(* LS Electric XG5000 project: project3 *)
(* PLC LSPLC *)

FUNCTION_BLOCK 위치사용
VAR_INPUT
    s11 : BOOL;
    s12 : BOOL;
    s13 : BOOL;
    s21 : BOOL;
    s22 : BOOL;
    s23 : BOOL;
    s31 : BOOL;
    s32 : BOOL;
    s33 : BOOL;
END_VAR
VAR_OUTPUT
    out11 : WORD;
    out12 : WORD;
    out13 : WORD;
    out21 : WORD;
    out22 : WORD;
    out23 : WORD;
    out31 : WORD;
    out32 : WORD;
    out33 : WORD;
END_VAR
VAR
    mout11 : INT;
    mout12 : INT;
    mout13 : INT;
    mout21 : INT;
    mout22 : INT;
    mout23 : INT;
    mout31 : INT;
    mout32 : INT;
    mout33 : INT;
END_VAR
VAR
    _e1 : R_TRIG;
    _e2 : F_TRIG;
    _e3 : R_TRIG;
    _e4 : F_TRIG;
    _e5 : R_TRIG;
    _e6 : F_TRIG;
    _e7 : R_TRIG;
    _e8 : F_TRIG;
    _e9 : R_TRIG;
    _e10 : F_TRIG;
    _e11 : R_TRIG;
    _e12 : F_TRIG;
    _e13 : R_TRIG;
    _e14 : F_TRIG;
    _e15 : R_TRIG;
    _e16 : F_TRIG;
    _e17 : R_TRIG;
    _e18 : F_TRIG;
END_VAR

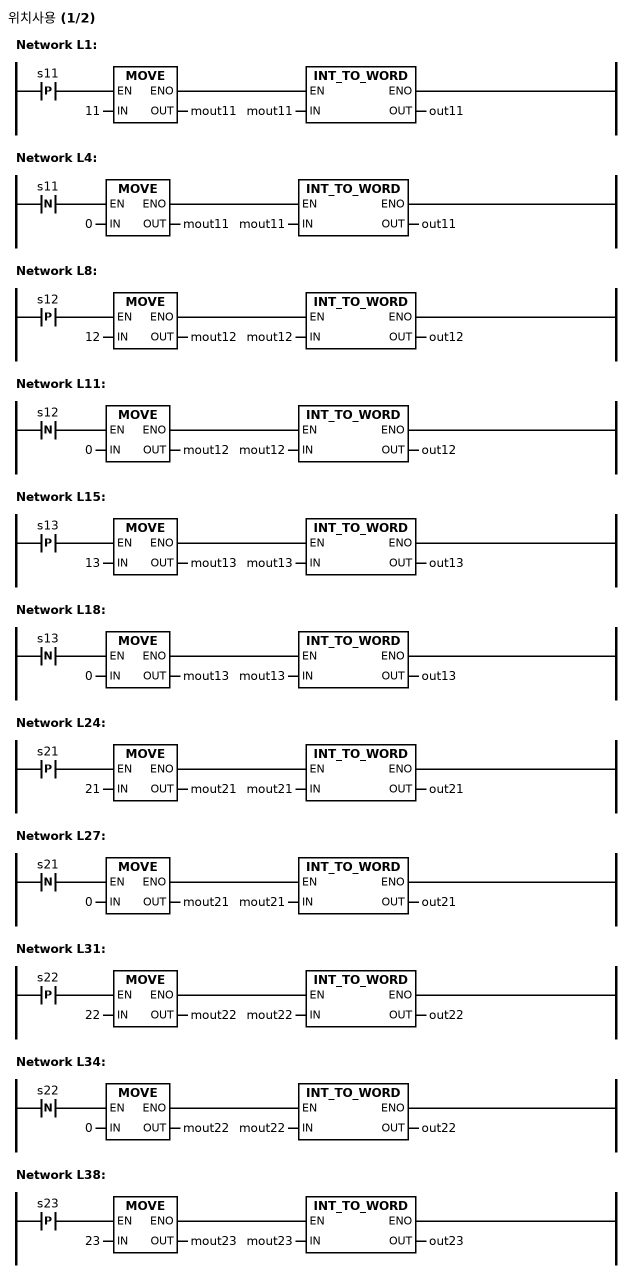
(* Rung L1 *)
_e1(CLK := s11);
IF _e1.Q THEN
    mout11 := 11;
    out11 := INT_TO_WORD(mout11);
END_IF;
(* Rung L4 *)
_e2(CLK := s11);
IF _e2.Q THEN
    mout11 := 0;
    out11 := INT_TO_WORD(mout11);
END_IF;
(* Rung L8 *)
_e3(CLK := s12);
IF _e3.Q THEN
    mout12 := 12;
    out12 := INT_TO_WORD(mout12);
END_IF;
(* Rung L11 *)
_e4(CLK := s12);
IF _e4.Q THEN
    mout12 := 0;
    out12 := INT_TO_WORD(mout12);
END_IF;
(* Rung L15 *)
_e5(CLK := s13);
IF _e5.Q THEN
    mout13 := 13;
    out13 := INT_TO_WORD(mout13);
END_IF;
(* Rung L18 *)
_e6(CLK := s13);
IF _e6.Q THEN
    mout13 := 0;
    out13 := INT_TO_WORD(mout13);
END_IF;
(* Rung L24 *)
_e7(CLK := s21);
IF _e7.Q THEN
    mout21 := 21;
    out21 := INT_TO_WORD(mout21);
END_IF;
(* Rung L27 *)
_e8(CLK := s21);
IF _e8.Q THEN
    mout21 := 0;
    out21 := INT_TO_WORD(mout21);
END_IF;
(* Rung L31 *)
_e9(CLK := s22);
IF _e9.Q THEN
    mout22 := 22;
    out22 := INT_TO_WORD(mout22);
END_IF;
(* Rung L34 *)
_e10(CLK := s22);
IF _e10.Q THEN
    mout22 := 0;
    out22 := INT_TO_WORD(mout22);
END_IF;
(* Rung L38 *)
_e11(CLK := s23);
IF _e11.Q THEN
    mout23 := 23;
    out23 := INT_TO_WORD(mout23);
END_IF;

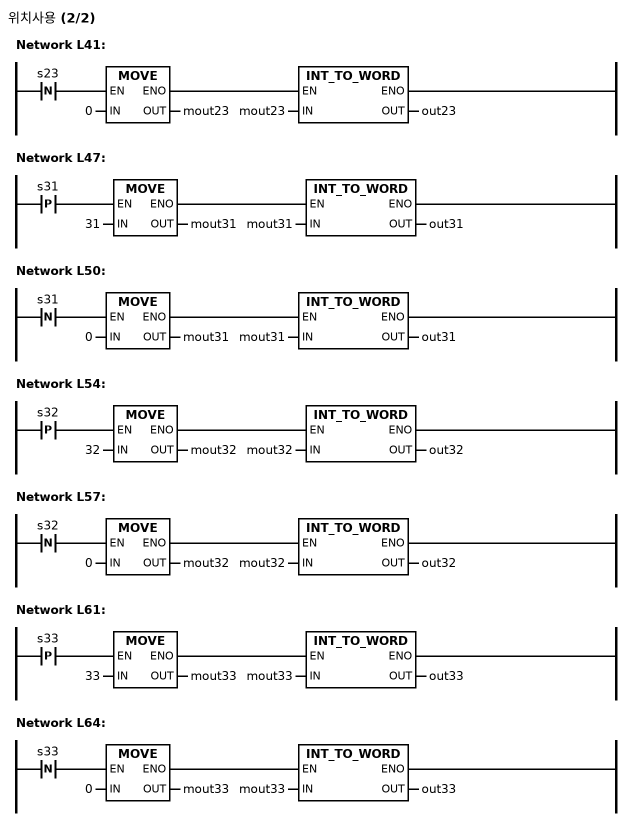
(* Rung L41 *)
_e12(CLK := s23);
IF _e12.Q THEN
    mout23 := 0;
    out23 := INT_TO_WORD(mout23);
END_IF;
(* Rung L47 *)
_e13(CLK := s31);
IF _e13.Q THEN
    mout31 := 31;
    out31 := INT_TO_WORD(mout31);
END_IF;
(* Rung L50 *)
_e14(CLK := s31);
IF _e14.Q THEN
    mout31 := 0;
    out31 := INT_TO_WORD(mout31);
END_IF;
(* Rung L54 *)
_e15(CLK := s32);
IF _e15.Q THEN
    mout32 := 32;
    out32 := INT_TO_WORD(mout32);
END_IF;
(* Rung L57 *)
_e16(CLK := s32);
IF _e16.Q THEN
    mout32 := 0;
    out32 := INT_TO_WORD(mout32);
END_IF;
(* Rung L61 *)
_e17(CLK := s33);
IF _e17.Q THEN
    mout33 := 33;
    out33 := INT_TO_WORD(mout33);
END_IF;
(* Rung L64 *)
_e18(CLK := s33);
IF _e18.Q THEN
    mout33 := 0;
    out33 := INT_TO_WORD(mout33);
END_IF;
END_FUNCTION_BLOCK

FUNCTION_BLOCK 초기화
VAR_INPUT
    초기화 : BOOL;
END_VAR
VAR_OUTPUT
    출력 : BOOL;
END_VAR
VAR
    INST1 : TON;
    INST2 : TP;
END_VAR

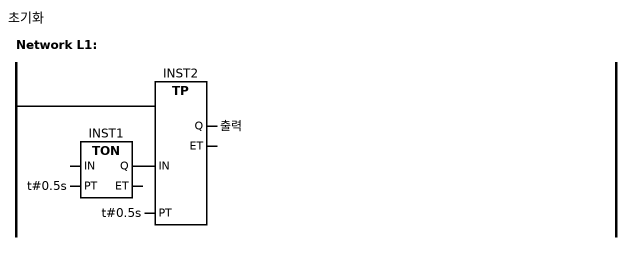
(* Rung L1 *)
INST1(IN := TRUE, PT := t#0.5s);
INST2(IN := INST1.Q, PT := t#0.5s, Q => 출력);
END_FUNCTION_BLOCK

FUNCTION_BLOCK move11
VAR_INPUT
    auto : BOOL;
END_VAR
VAR_OUTPUT
    move11 : BOOL; (* 11 *)
    move21 : BOOL; (* 21 *)
    move31 : BOOL; (* 31 *)
    move32 : BOOL; (* 32 *)
    move33 : BOOL; (* 33 *)
END_VAR
VAR
    X1 : TON;
    X2 : TON;
    X3 : TON;
    Y1 : TON;
    Y2 : TON;
END_VAR

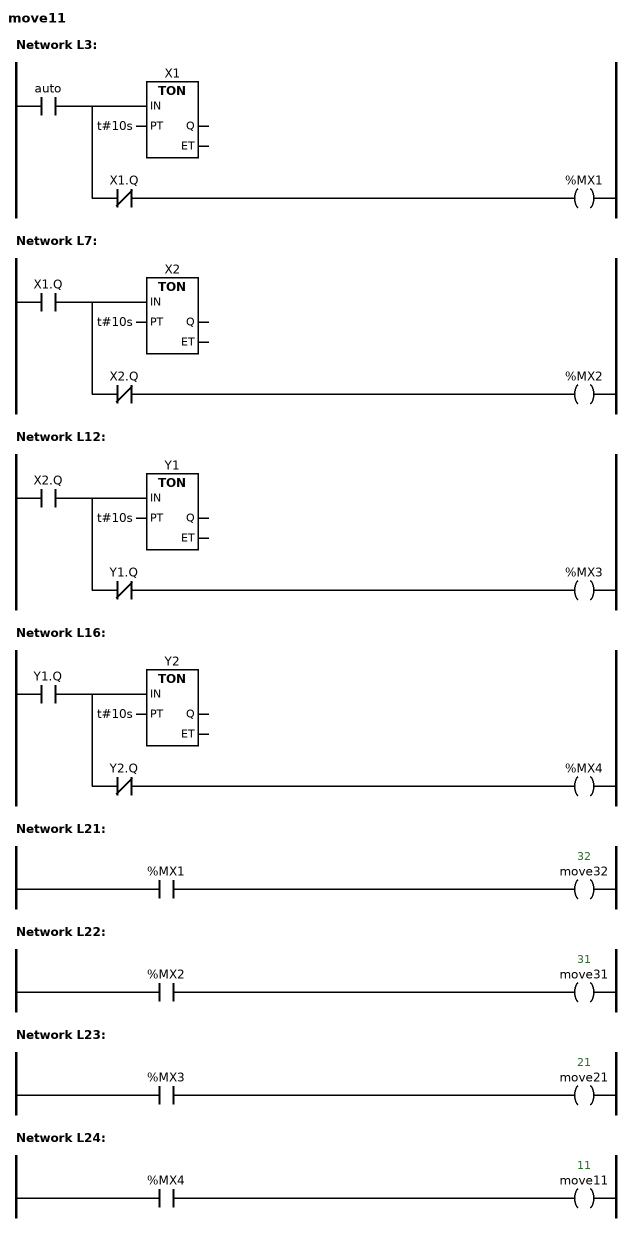
(* Rung L3 *)
X1(IN := auto, PT := t#10s);
%MX1 := auto AND NOT X1.Q;
(* Rung L7 *)
X2(IN := X1.Q, PT := t#10s);
%MX2 := X1.Q AND NOT X2.Q;
(* Rung L12 *)
Y1(IN := X2.Q, PT := t#10s);
%MX3 := X2.Q AND NOT Y1.Q;
(* Rung L16 *)
Y2(IN := Y1.Q, PT := t#10s);
%MX4 := Y1.Q AND NOT Y2.Q;
(* Rung L21 *)
move32 := %MX1;
(* Rung L22 *)
move31 := %MX2;
(* Rung L23 *)
move21 := %MX3;
(* Rung L24 *)
move11 := %MX4;
END_FUNCTION_BLOCK

FUNCTION_BLOCK move12
VAR_INPUT
    auto : BOOL;
END_VAR
VAR
    move12 : BOOL; (* 12 *)
    move22 : BOOL; (* 22 *)
    move32 : BOOL; (* 32 *)
    X1 : TON;
    X2 : TON;
    Y1 : TON;
    Y2 : TON;
END_VAR

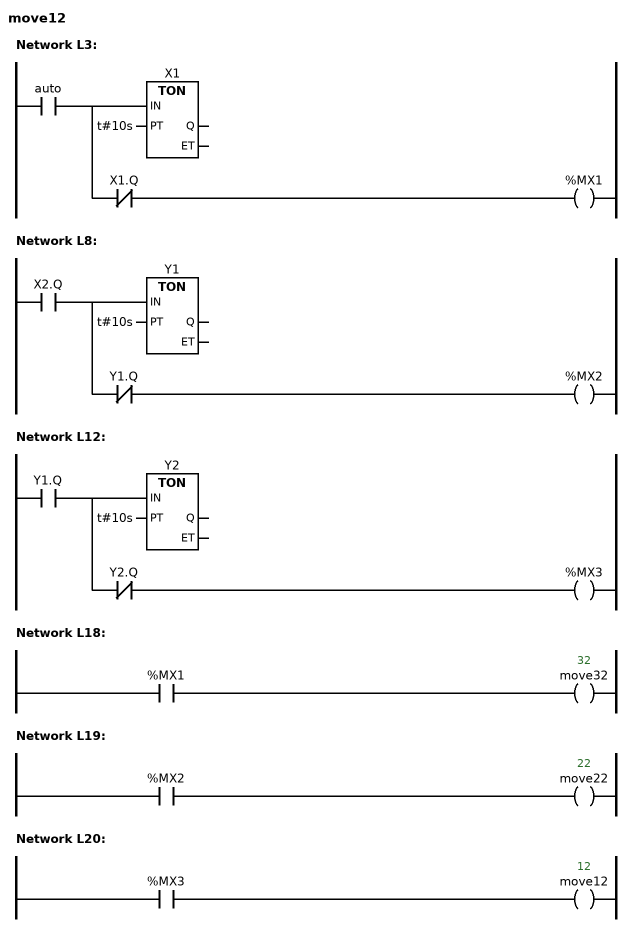
(* Rung L3 *)
X1(IN := auto, PT := t#10s);
%MX1 := auto AND NOT X1.Q;
(* Rung L8 *)
Y1(IN := X2.Q, PT := t#10s);
%MX2 := X2.Q AND NOT Y1.Q;
(* Rung L12 *)
Y2(IN := Y1.Q, PT := t#10s);
%MX3 := Y1.Q AND NOT Y2.Q;
(* Rung L18 *)
move32 := %MX1;
(* Rung L19 *)
move22 := %MX2;
(* Rung L20 *)
move12 := %MX3;
END_FUNCTION_BLOCK

FUNCTION_BLOCK move13
VAR_INPUT
    auto : BOOL;
END_VAR
VAR_OUTPUT
    move33 : BOOL; (* 33 *)
    move32 : BOOL; (* 32 *)
    move22 : BOOL;
    move12 : BOOL;
END_VAR
VAR
    move13 : BOOL; (* 13 *)
    move23 : BOOL; (* 23 *)
    X1 : TON;
    X2 : TON;
    Y1 : TON;
    Y2 : TON;
END_VAR

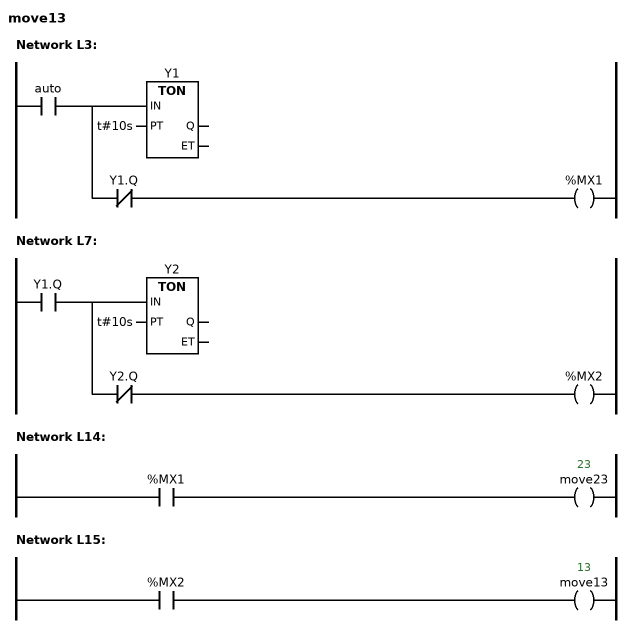
(* Rung L3 *)
Y1(IN := auto, PT := t#10s);
%MX1 := auto AND NOT Y1.Q;
(* Rung L7 *)
Y2(IN := Y1.Q, PT := t#10s);
%MX2 := Y1.Q AND NOT Y2.Q;
(* Rung L14 *)
move23 := %MX1;
(* Rung L15 *)
move13 := %MX2;
END_FUNCTION_BLOCK

PROGRAM NewProgram (* task: 스캔 프로그램 *)
VAR
    A AT %QX0.2.0 : BOOL;
    a1 : ARRAY[0..9] OF INT;
    AD : BOOL := 0;
    A_check AT %QX0.5.0 : BOOL;
    A_delay : TON;
    A_delay_유지 : BOOL;
    A_last : TON;
    A_pull : BOOL;
    A_push : BOOL;
    A_way AT %QX0.6.0 : BOOL;
    A단락 : BOOL;
    A센서 AT %QX0.9.0 : BOOL; (* 센서 *)
    A센서_딜레이 : TON;
    A센서상태변경 : TON;
    A센서지연 : TON;
    A센서지연1 : TON;
    A실린더_OFF AT %IX0.1.1 : BOOL; (* 실린더 *)
    A실린더_ON AT %IX0.1.0 : BOOL; (* 실린더 *)
    A지연 : TON;
    A차단 : TON;
    A카운트 : CTU_INT;
    A타이머 : TON;
    B AT %QX0.2.1 : BOOL;
    BD : BOOL := 0;
    B_check AT %QX0.5.1 : BOOL;
    B_delay : TON;
    B_delay_유지 : BOOL;
    B_last : TON;
    b_pull : BOOL;
    B_push : BOOL;
    B_way AT %QX0.6.1 : BOOL;
    B단락 : BOOL;
    B센서 AT %QX0.9.1 : BOOL; (* 센서 *)
    B센서_딜레이 : TON;
    B센서상태변경 : TON;
    B센서지연 : TON;
    B센서지연1 : TON;
    B실린더_OFF AT %IX0.1.3 : BOOL; (* 실린더 *)
    B실린더_ON AT %IX0.1.2 : BOOL; (* 실린더 *)
    B지연 : TON;
    B차단 : TON;
    B카운트 : CTU_INT;
    B타이머 : TON;
    C AT %QX0.2.2 : BOOL;
    CD : BOOL := 0;
    CU : BOOL;
    C_check AT %QX0.5.2 : BOOL;
    C_delay : TON;
    C_delay_유지 : BOOL;
    C_last : TON;
    c_out : BOOL;
    C_pull : BOOL;
    C_push : BOOL;
    C_way AT %QX0.6.2 : BOOL;
    C단락 : BOOL;
    C센서 AT %QX0.9.2 : BOOL; (* 센서 *)
    C센서_딜레이 : TON;
    C센서상태변경 : TON;
    C센서지연 : TON;
    C센서지연1 : TON;
    C실린더_OFF AT %IX0.1.5 : BOOL; (* 실린더 *)
    C실린더_ON AT %IX0.1.4 : BOOL; (* 실린더 *)
    C지연 : TON;
    C차단 : TON;
    C카운트 : CTUD_INT;
    C카운트1 : CTUD_INT;
    C타이머 : TON;
    C타이머1 : TON;
    C타이머2 : TON;
    D1 : WORD;
    D91 : TIME;
    delay : TP;
    done : BOOL;
    d_a AT %IW0.3.0 : WORD;
    d_a_out : UDINT;
    d_a_time : TIME;
    d_b AT %IW0.3.1 : WORD;
    d_b_out : UDINT;
    d_b_time : TIME;
    d_input : BOOL;
    ET : TIME;
    fifo : FIFO_INT;
    INST : TP;
    INST1 : TP;
    INST10 : TP;
    INST11 : TP;
    INST12 : TP;
    INST13 : TP;
    INST14 : TP;
    INST15 : TP;
    INST16 : TP;
    INST17 : TP;
    INST18 : TP;
    INST19 : TP;
    INST2 : TP;
    INST20 : TP;
    INST21 : TP;
    INST22 : TP;
    INST23 : TP;
    INST24 : TP;
    INST25 : TP;
    INST26 : TP;
    INST27 : TP;
    INST28 : TP;
    INST29 : TP;
    INST3 : TP;
    INST30 : TP;
    INST31 : TP;
    INST32 : TP;
    INST33 : TP;
    INST34 : TP;
    INST35 : TP;
    INST36 : TP;
    INST37 : TP;
    INST38 : CTUD_INT;
    INST4 : TP;
    INST5 : TP;
    INST6 : TP;
    INST7 : TP;
    INST8 : TP;
    INST9 : TP;
    LD : BOOL;
    LOAD : BOOL;
    OUT AT %QW0.8.0 : INT;
    output1 : INT;
    output2 : UDINT;
    output3 : INT;
    output4 : UDINT;
    output5 : INT;
    output6 : UDINT;
    output7 : INT;
    output8 : UDINT;
    prev AT %QW0.8.1 : WORD;
    prev_int : INT;
    PV : INT;
    QD : BOOL;
    QU : BOOL;
    R : BOOL;
    rand : INT;
    reset : BOOL;
    RST : BOOL;
    s11 : BOOL;
    s12 : BOOL;
    s13 : BOOL;
    s21 : BOOL;
    s22 : BOOL;
    s23 : BOOL;
    s31 : BOOL;
    s32 : BOOL;
    s33 : BOOL;
    set : BOOL;
    signal : BOOL;
    stack : CTUD_INT;
    stack_max : INT := 9; (* max *)
    stack_센서 : BOOL;
    stack센서 : BOOL;
    start : BOOL;
    stop AT %IX0.0.1 : BOOL;
    system_on AT %IX0.0.0 : BOOL;
    temp AT %IX0.0.2 : BOOL;
    test1 : BOOL;
    test2 : BOOL;
    three : WORD := 3;
    time1 : TIME;
    time2 : TIME;
    time3 : TIME;
    time4 : TIME;
    UNLD : BOOL;
    X1 : TON;
    X2 : TON;
    X3 : TON;
    Y1 : TON;
    Y2 : TON;
    Y3 : TON;
    _T15S : BOOL;
    긴급제동 : BOOL; (* RED *)
    난수1 : TON;
    난수2 : TON;
    난수회로차단 : TP;
    놓기 AT %QX0.0.49 : BOOL;
    단선 AT %QX0.8.1 : BOOL;
    도착 AT %QX0.5.3 : BOOL;
    딜레이 : TON;
    랜덤수 : INT;
    명령 : BOOL;
    물품없음 : BOOL; (* WHITE *)
    반시계 AT %QX0.0.62 : BOOL;
    백색등 : BOOL;
    상 AT %QX0.0.60 : BOOL;
    선택값 : INT;
    소요시간1 : TIME;
    수동 : BOOL;
    순환값 : WORD;
    숫자 : INT := 1;
    시계 AT %QX0.0.61 : BOOL;
    시퀀스1 AT %MW4 : INT;
    시퀀스2 AT %MW8 : INT;
    신호 AT %QX0.6.3 : BOOL;
    앞 AT %QX0.0.59 : BOOL;
    연기 : BOOL;
    위치사용 : 위치사용;
    임시 : BOOL;
    입고 : CTUD_INT;
    입력 : BOOL;
    입력1 AT %QX0.6.4 : BOOL;
    입력시간1 AT %MW6 : INT;
    입력시간2 AT %MW2 : INT;
    입력시간3 AT %MW10 : INT;
    입력시간4 AT %MW12 : INT;
    입력신호 AT %QW0.6.3 : INT;
    자동 : BOOL;
    잡기 AT %QX0.0.63 : BOOL;
    저장 : FIFO_INT;
    정상가동 : BOOL; (* GREEN *)
    지연 : TON;
    지연1 : TP;
    초기화 : 초기화;
    출력 : BOOL;
    칸1 AT %QX0.0.50 : BOOL;
    칸10 AT %QX0.0.44 : BOOL;
    칸11 AT %QX0.0.47 : BOOL;
    칸12 AT %QX0.0.46 : BOOL;
    칸2 AT %QX0.0.51 : BOOL;
    칸3 AT %QX0.0.52 : BOOL;
    칸4 AT %QX0.0.53 : BOOL;
    칸5 AT %QX0.0.54 : BOOL;
    칸6 AT %QX0.0.55 : BOOL;
    칸7 AT %QX0.0.56 : BOOL;
    칸8 AT %QX0.0.57 : BOOL;
    칸9 AT %QX0.0.58 : BOOL;
    컨베이어벨트 AT %QX0.4.4 : BOOL;
    컨베이어타이머 : TON;
    하 AT %QX0.0.45 : BOOL;
    하나출력 : BOOL;
END_VAR
VAR
    _t1 : BOOL;
    _e2 : R_TRIG;
    _e3 : F_TRIG;
    _e4 : F_TRIG;
    _e5 : F_TRIG;
    _e6 : F_TRIG;
    _e7 : R_TRIG;
    _e8 : R_TRIG;
    _p9 : BOOL;
    _p10 : BOOL;
    _e11 : R_TRIG;
    _p12 : BOOL;
    _p13 : BOOL;
    _e14 : R_TRIG;
    _p15 : BOOL;
    _p16 : BOOL;
    _e17 : R_TRIG;
    _p18 : BOOL;
    _e19 : R_TRIG;
    _e20 : R_TRIG;
    _e21 : R_TRIG;
    _t22 : BOOL;
    _e23 : F_TRIG;
    _e24 : F_TRIG;
    _e25 : F_TRIG;
    _e26 : F_TRIG;
    _e27 : F_TRIG;
    _e28 : F_TRIG;
    _e29 : F_TRIG;
    _e30 : F_TRIG;
    _e31 : F_TRIG;
    _e32 : F_TRIG;
    _e33 : F_TRIG;
    _e34 : F_TRIG;
    _e35 : F_TRIG;
    _e36 : F_TRIG;
    _e37 : F_TRIG;
    _e38 : F_TRIG;
    _e39 : F_TRIG;
    _e40 : F_TRIG;
    _e41 : F_TRIG;
    _e42 : F_TRIG;
    _e43 : F_TRIG;
    _e44 : F_TRIG;
    _e45 : F_TRIG;
    _e46 : F_TRIG;
    _e47 : F_TRIG;
    _e48 : F_TRIG;
    _e49 : F_TRIG;
    _e50 : F_TRIG;
    _e51 : F_TRIG;
    _e52 : F_TRIG;
    _e53 : F_TRIG;
    _e54 : F_TRIG;
    _e55 : F_TRIG;
    _e56 : F_TRIG;
    _e57 : F_TRIG;
    _e58 : F_TRIG;
    _e59 : F_TRIG;
    _e60 : F_TRIG;
    _e61 : F_TRIG;
END_VAR

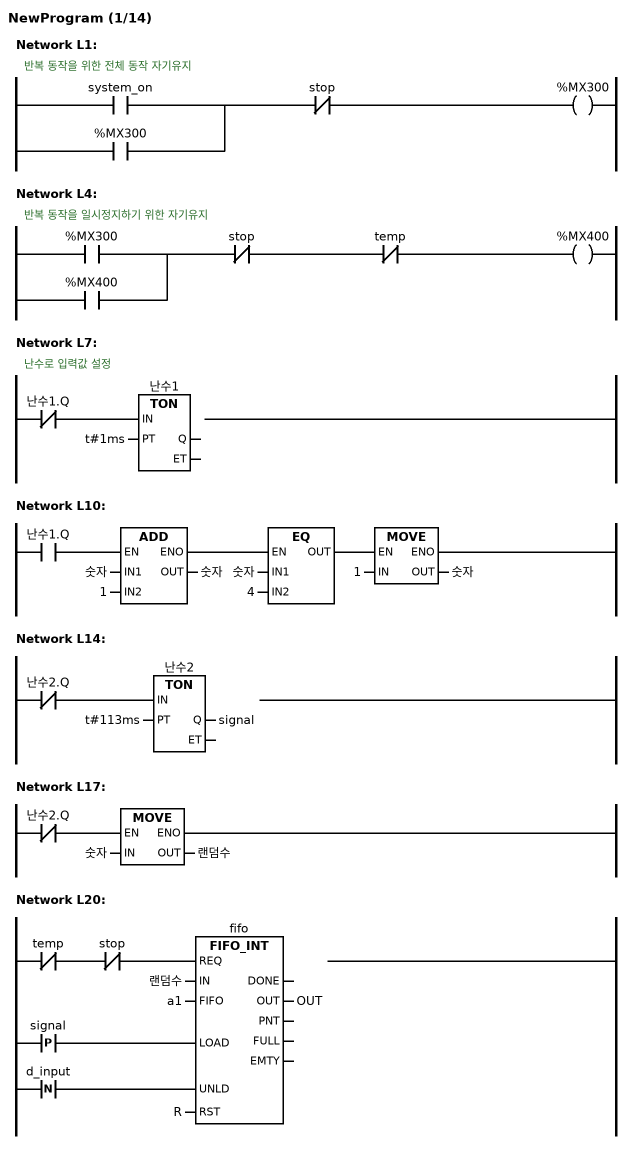
(* 반복 동작을 위한 전체 동작 자기유지 *)
(* Rung L1 *)
%MX300 := (system_on OR %MX300) AND NOT stop;
(* 반복 동작을 일시정지하기 위한 자기유지 *)
(* Rung L4 *)
%MX400 := (%MX300 OR %MX400) AND NOT stop AND NOT temp;
(* 난수로 입력값 설정 *)
(* Rung L7 *)
난수1(IN := NOT 난수1.Q, PT := t#1ms);
(* Rung L10 *)
IF 난수1.Q THEN
    숫자 := 숫자 + 1;
    _t1 := 숫자 = 4;
END_IF;
IF _t1 THEN 숫자 := 1; END_IF;
(* Rung L14 *)
난수2(IN := NOT 난수2.Q, PT := t#113ms, Q => signal);
(* Rung L17 *)
IF NOT 난수2.Q THEN 랜덤수 := 숫자; END_IF;
(* Rung L20 *)
_e2(CLK := signal);
_e3(CLK := d_input);
fifo(REQ := NOT temp AND NOT stop, IN := 랜덤수, FIFO := a1, LOAD := _e2.Q, UNLD := _e3.Q, RST := R, OUT => OUT);

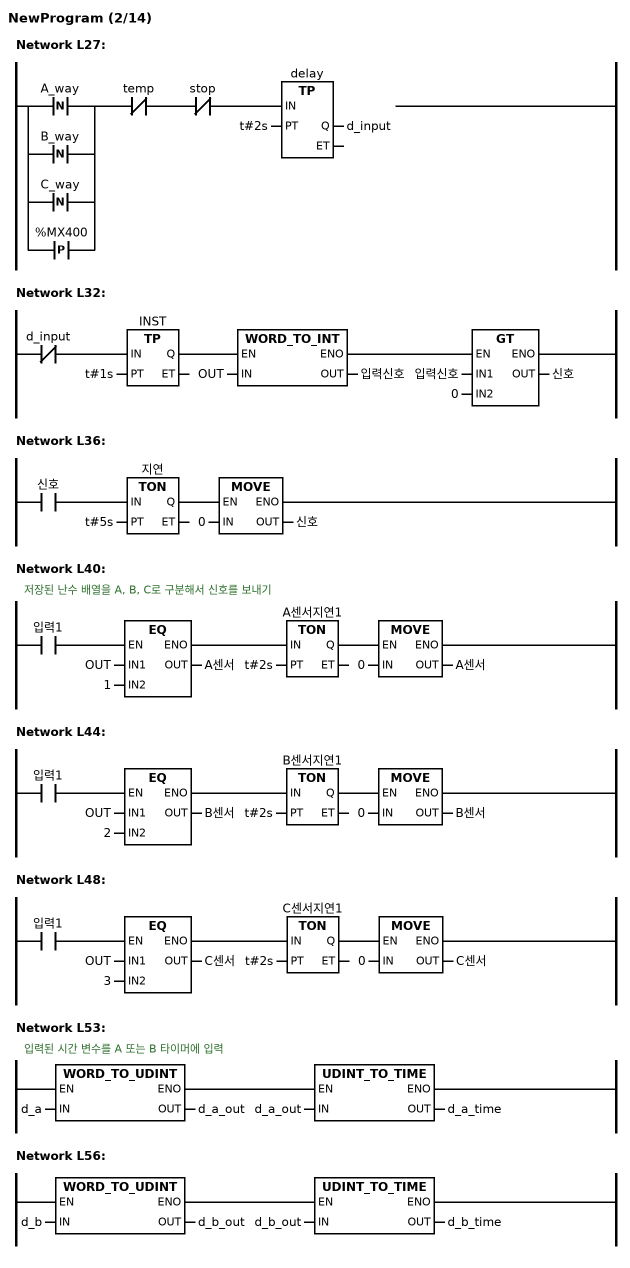
(* Rung L27 *)
_e4(CLK := A_way);
_e5(CLK := B_way);
_e6(CLK := C_way);
_e7(CLK := %MX400);
delay(IN := (_e4.Q OR _e5.Q OR _e6.Q OR _e7.Q) AND NOT temp AND NOT stop, PT := t#2s, Q => d_input);
(* Rung L32 *)
INST(IN := NOT d_input, PT := t#1s);
IF INST.Q THEN
    입력신호 := WORD_TO_INT(OUT);
    신호 := 입력신호 > 0;
END_IF;
(* Rung L36 *)
지연(IN := 신호, PT := t#5s);
IF 지연.Q THEN 신호 := 0; END_IF;
(* 저장된 난수 배열을 A, B, C로 구분해서 신호를 보내기 *)
(* Rung L40 *)
IF 입력1 THEN A센서 := OUT = 1; END_IF;
A센서지연1(IN := 입력1, PT := t#2s);
IF A센서지연1.Q THEN A센서 := 0; END_IF;
(* Rung L44 *)
IF 입력1 THEN B센서 := OUT = 2; END_IF;
B센서지연1(IN := 입력1, PT := t#2s);
IF B센서지연1.Q THEN B센서 := 0; END_IF;
(* Rung L48 *)
IF 입력1 THEN C센서 := OUT = 3; END_IF;
C센서지연1(IN := 입력1, PT := t#2s);
IF C센서지연1.Q THEN C센서 := 0; END_IF;
(* 입력된 시간 변수를 A 또는 B 타이머에 입력 *)
(* Rung L53 *)
d_a_out := WORD_TO_UDINT(d_a);
d_a_time := UDINT_TO_TIME(d_a_out);
(* Rung L56 *)
d_b_out := WORD_TO_UDINT(d_b);
d_b_time := UDINT_TO_TIME(d_b_out);

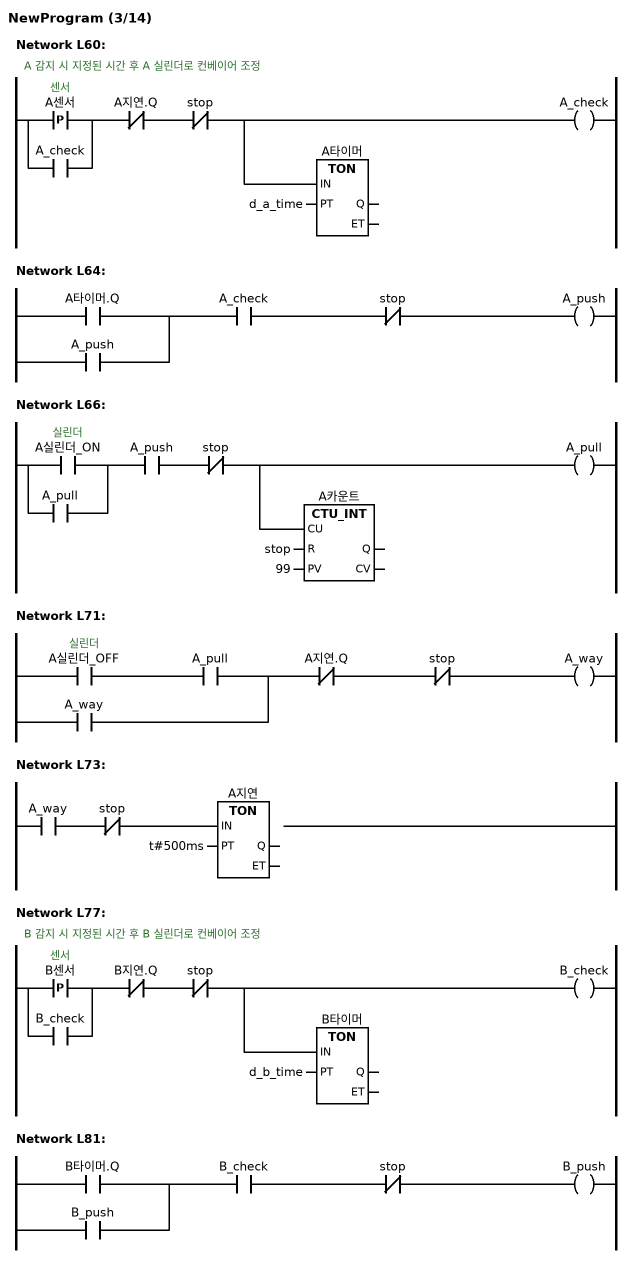
(* A 감지 시 지정된 시간 후 A 실린더로 컨베이어 조정 *)
(* Rung L60 *)
_e8(CLK := A센서);
_p9 := (_e8.Q OR A_check) AND NOT A지연.Q AND NOT stop;
A_check := _p9;
A타이머(IN := _p9, PT := d_a_time);
(* Rung L64 *)
A_push := (A타이머.Q OR A_push) AND A_check AND NOT stop;
(* Rung L66 *)
_p10 := (A실린더_ON OR A_pull) AND A_push AND NOT stop;
A_pull := _p10;
A카운트(CU := _p10, R := stop, PV := 99);
(* Rung L71 *)
A_way := ((A실린더_OFF AND A_pull) OR A_way) AND NOT A지연.Q AND NOT stop;
(* Rung L73 *)
A지연(IN := A_way AND NOT stop, PT := t#500ms);
(* B 감지 시 지정된 시간 후 B 실린더로 컨베이어 조정 *)
(* Rung L77 *)
_e11(CLK := B센서);
_p12 := (_e11.Q OR B_check) AND NOT B지연.Q AND NOT stop;
B_check := _p12;
B타이머(IN := _p12, PT := d_b_time);
(* Rung L81 *)
B_push := (B타이머.Q OR B_push) AND B_check AND NOT stop;

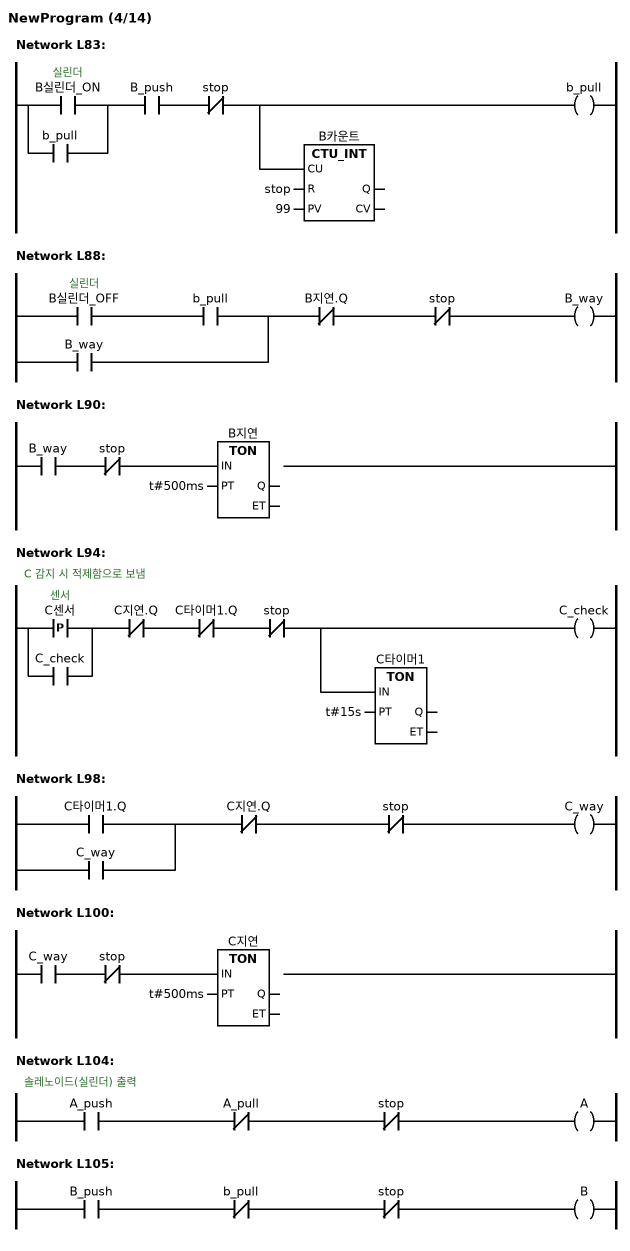
(* Rung L83 *)
_p13 := (B실린더_ON OR b_pull) AND B_push AND NOT stop;
b_pull := _p13;
B카운트(CU := _p13, R := stop, PV := 99);
(* Rung L88 *)
B_way := ((B실린더_OFF AND b_pull) OR B_way) AND NOT B지연.Q AND NOT stop;
(* Rung L90 *)
B지연(IN := B_way AND NOT stop, PT := t#500ms);
(* C 감지 시 적제함으로 보냄 *)
(* Rung L94 *)
_e14(CLK := C센서);
_p15 := (_e14.Q OR C_check) AND NOT C지연.Q AND NOT C타이머1.Q AND NOT stop;
C_check := _p15;
C타이머1(IN := _p15, PT := t#15s);
(* Rung L98 *)
C_way := (C타이머1.Q OR C_way) AND NOT C지연.Q AND NOT stop;
(* Rung L100 *)
C지연(IN := C_way AND NOT stop, PT := t#500ms);
(* 솔레노이드(실린더) 출력 *)
(* Rung L104 *)
A := A_push AND NOT A_pull AND NOT stop;
(* Rung L105 *)
B := B_push AND NOT b_pull AND NOT stop;

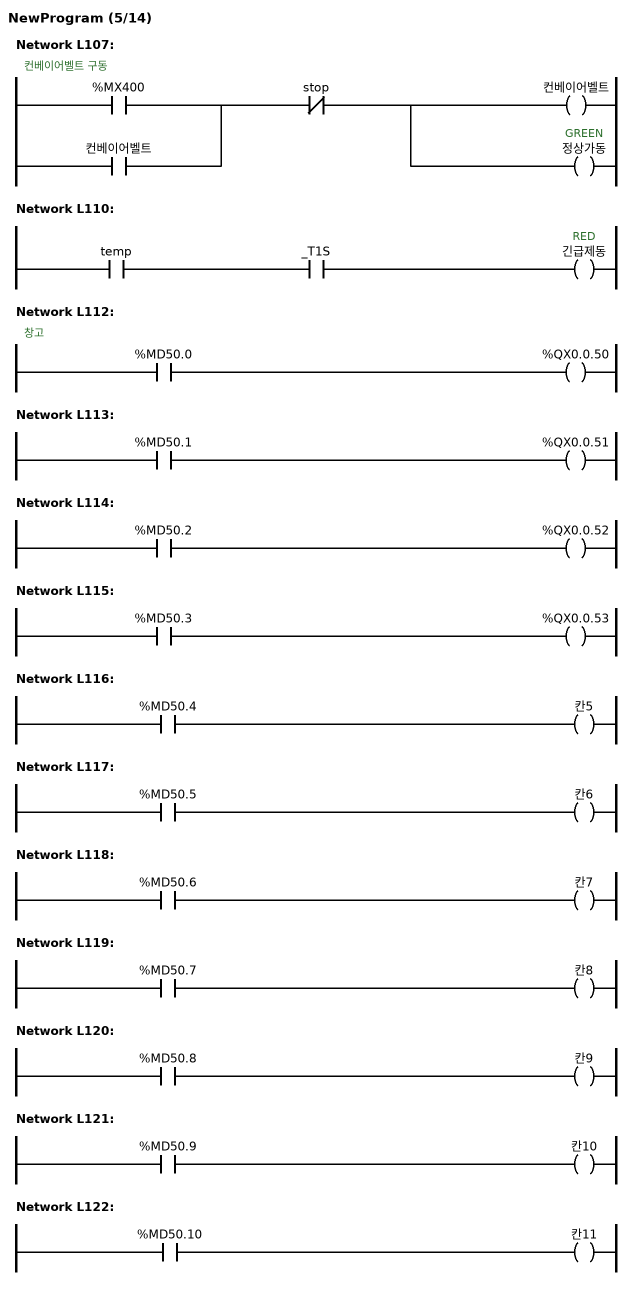
(* 컨베이어벨트 구동 *)
(* Rung L107 *)
_p16 := (%MX400 OR 컨베이어벨트) AND NOT stop;
컨베이어벨트 := _p16;
정상가동 := _p16;
(* Rung L110 *)
긴급제동 := temp AND _T1S;
(* 창고 *)
(* Rung L112 *)
%QX0.0.50 := %MD50.0;
(* Rung L113 *)
%QX0.0.51 := %MD50.1;
(* Rung L114 *)
%QX0.0.52 := %MD50.2;
(* Rung L115 *)
%QX0.0.53 := %MD50.3;
(* Rung L116 *)
칸5 := %MD50.4;
(* Rung L117 *)
칸6 := %MD50.5;
(* Rung L118 *)
칸7 := %MD50.6;
(* Rung L119 *)
칸8 := %MD50.7;
(* Rung L120 *)
칸9 := %MD50.8;
(* Rung L121 *)
칸10 := %MD50.9;
(* Rung L122 *)
칸11 := %MD50.10;

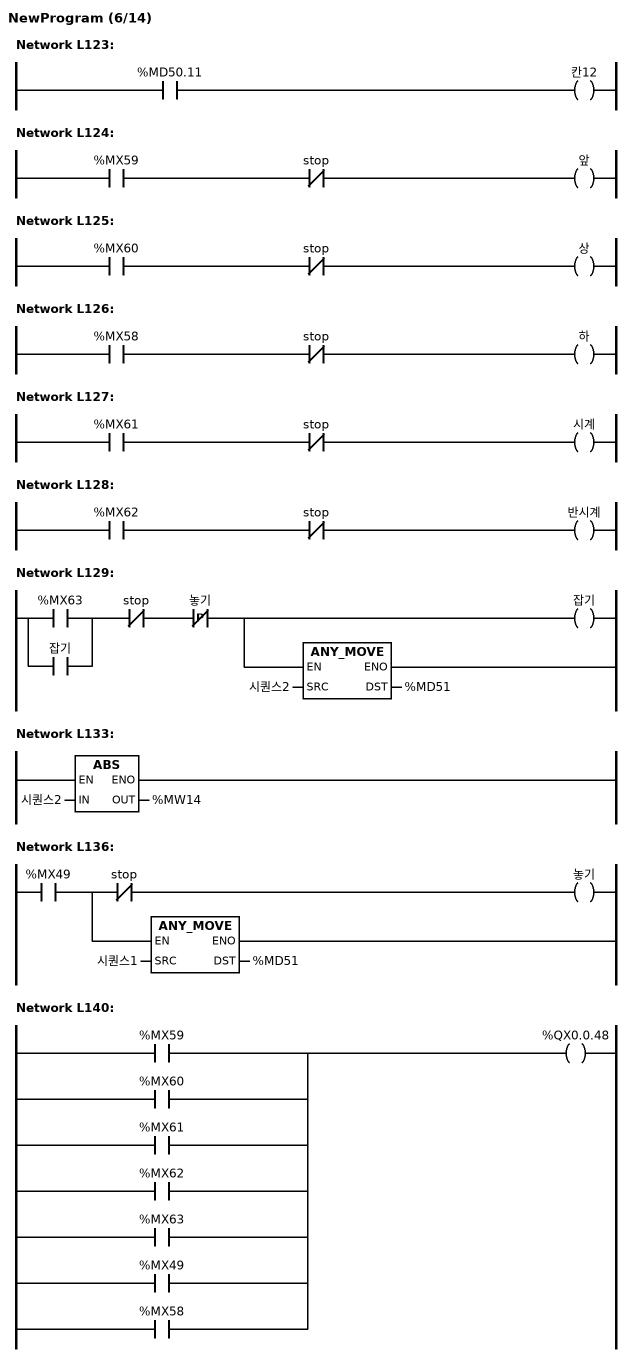
(* Rung L123 *)
칸12 := %MD50.11;
(* Rung L124 *)
앞 := %MX59 AND NOT stop;
(* Rung L125 *)
상 := %MX60 AND NOT stop;
(* Rung L126 *)
하 := %MX58 AND NOT stop;
(* Rung L127 *)
시계 := %MX61 AND NOT stop;
(* Rung L128 *)
반시계 := %MX62 AND NOT stop;
(* Rung L129 *)
_e17(CLK := 놓기);
_p18 := (%MX63 OR 잡기) AND NOT stop AND NOT _e17.Q;
잡기 := _p18;
IF _p18 THEN %MD51 := ANY_MOVE(SRC := 시퀀스2); END_IF;
(* Rung L133 *)
%MW14 := ABS(시퀀스2);
(* Rung L136 *)
놓기 := %MX49 AND NOT stop;
IF %MX49 THEN %MD51 := ANY_MOVE(SRC := 시퀀스1); END_IF;
(* Rung L140 *)
%QX0.0.48 := %MX59 OR %MX60 OR %MX61 OR %MX62 OR %MX63 OR %MX49 OR %MX58;

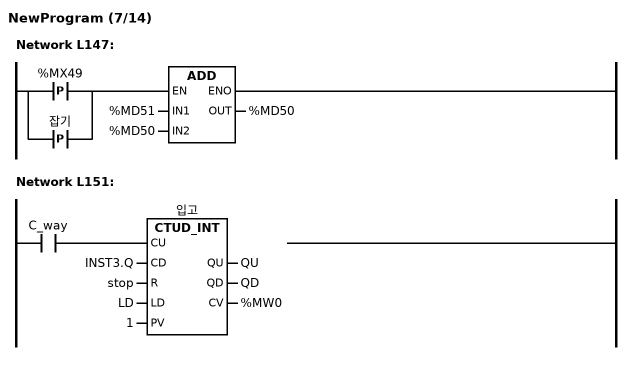
(* Rung L147 *)
_e19(CLK := %MX49);
_e20(CLK := 잡기);
IF _e19.Q OR _e20.Q THEN %MD50 := %MD51 + %MD50; END_IF;
(* Rung L151 *)
입고(CU := C_way, CD := INST3.Q, R := stop, LD := LD, PV := 1, QU => QU, QD => QD, CV => %MW0);

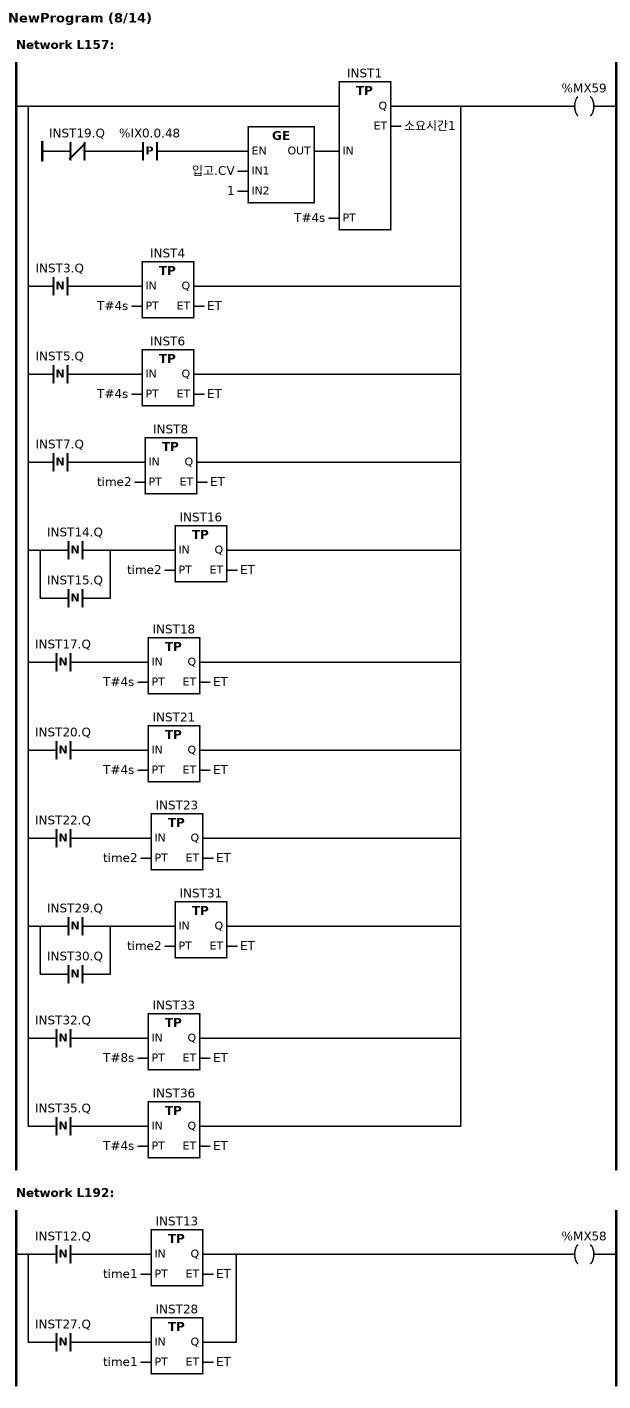
(* Rung L157 *)
_e21(CLK := %IX0.0.48);
IF NOT INST19.Q AND _e21.Q THEN _t22 := 입고.CV >= 1; END_IF;
INST1(IN := _t22, PT := T#4s, ET => 소요시간1);
_e23(CLK := INST3.Q);
INST4(IN := _e23.Q, PT := T#4s, ET => ET);
_e24(CLK := INST5.Q);
INST6(IN := _e24.Q, PT := T#4s, ET => ET);
_e25(CLK := INST7.Q);
INST8(IN := _e25.Q, PT := time2, ET => ET);
_e26(CLK := INST14.Q);
_e27(CLK := INST15.Q);
INST16(IN := _e26.Q OR _e27.Q, PT := time2, ET => ET);
_e28(CLK := INST17.Q);
INST18(IN := _e28.Q, PT := T#4s, ET => ET);
_e29(CLK := INST20.Q);
INST21(IN := _e29.Q, PT := T#4s, ET => ET);
_e30(CLK := INST22.Q);
INST23(IN := _e30.Q, PT := time2, ET => ET);
_e31(CLK := INST29.Q);
_e32(CLK := INST30.Q);
INST31(IN := _e31.Q OR _e32.Q, PT := time2, ET => ET);
_e33(CLK := INST32.Q);
INST33(IN := _e33.Q, PT := T#8s, ET => ET);
_e34(CLK := INST35.Q);
INST36(IN := _e34.Q, PT := T#4s, ET => ET);
%MX59 := INST1.Q OR INST4.Q OR INST6.Q OR INST8.Q OR INST16.Q OR INST18.Q OR INST21.Q OR INST23.Q OR INST31.Q OR INST33.Q OR INST36.Q;
(* Rung L192 *)
_e35(CLK := INST12.Q);
INST13(IN := _e35.Q, PT := time1, ET => ET);
_e36(CLK := INST27.Q);
INST28(IN := _e36.Q, PT := time1, ET => ET);
%MX58 := INST13.Q OR INST28.Q;

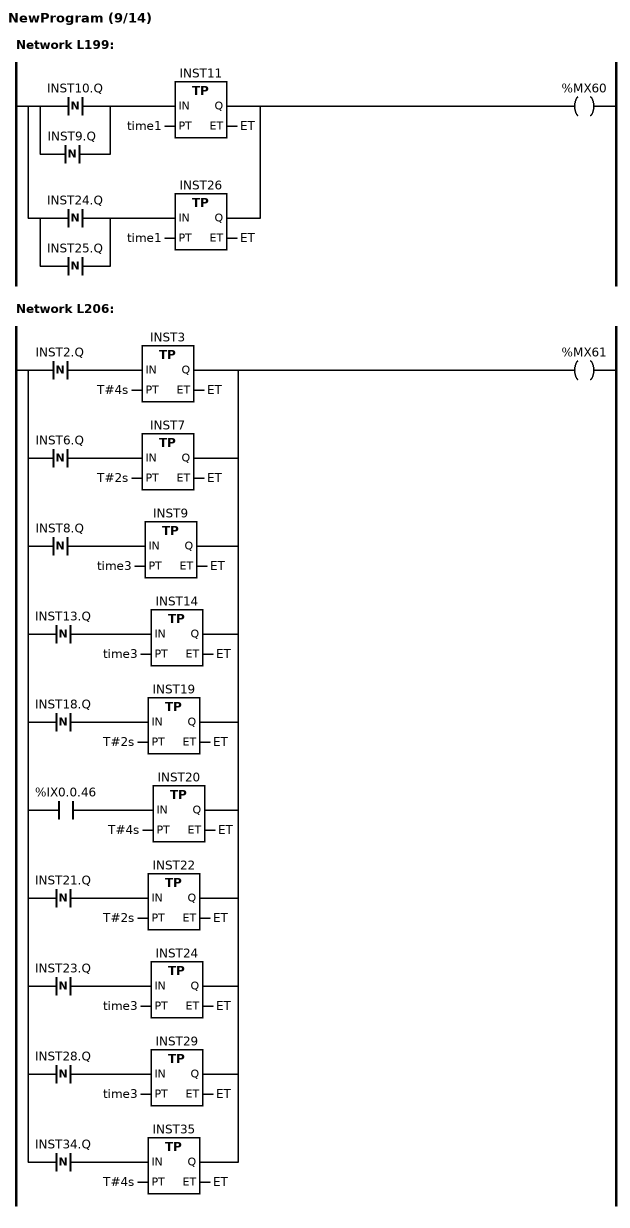
(* Rung L199 *)
_e37(CLK := INST10.Q);
_e38(CLK := INST9.Q);
INST11(IN := _e37.Q OR _e38.Q, PT := time1, ET => ET);
_e39(CLK := INST24.Q);
_e40(CLK := INST25.Q);
INST26(IN := _e39.Q OR _e40.Q, PT := time1, ET => ET);
%MX60 := INST11.Q OR INST26.Q;
(* Rung L206 *)
_e41(CLK := INST2.Q);
INST3(IN := _e41.Q, PT := T#4s, ET => ET);
_e42(CLK := INST6.Q);
INST7(IN := _e42.Q, PT := T#2s, ET => ET);
_e43(CLK := INST8.Q);
INST9(IN := _e43.Q, PT := time3, ET => ET);
_e44(CLK := INST13.Q);
INST14(IN := _e44.Q, PT := time3, ET => ET);
_e45(CLK := INST18.Q);
INST19(IN := _e45.Q, PT := T#2s, ET => ET);
INST20(IN := %IX0.0.46, PT := T#4s, ET => ET);
_e46(CLK := INST21.Q);
INST22(IN := _e46.Q, PT := T#2s, ET => ET);
_e47(CLK := INST23.Q);
INST24(IN := _e47.Q, PT := time3, ET => ET);
_e48(CLK := INST28.Q);
INST29(IN := _e48.Q, PT := time3, ET => ET);
_e49(CLK := INST34.Q);
INST35(IN := _e49.Q, PT := T#4s, ET => ET);
%MX61 := INST3.Q OR INST7.Q OR INST9.Q OR INST14.Q OR INST19.Q OR INST20.Q OR INST22.Q OR INST24.Q OR INST29.Q OR INST35.Q;

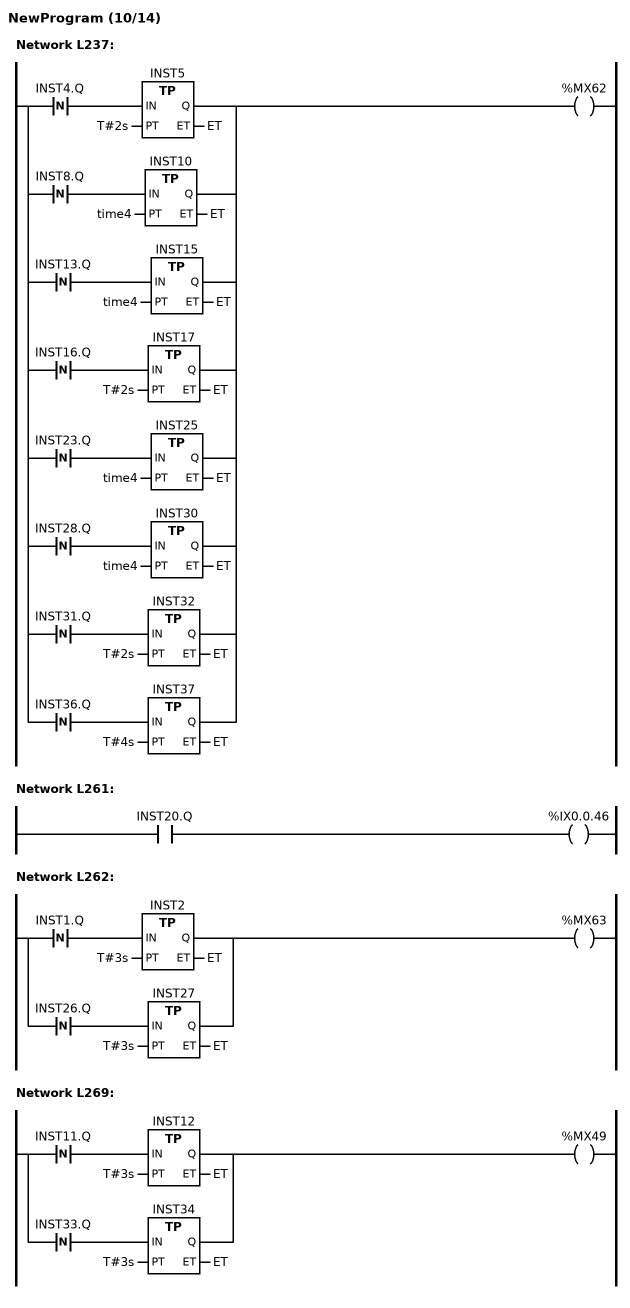
(* Rung L237 *)
_e50(CLK := INST4.Q);
INST5(IN := _e50.Q, PT := T#2s, ET => ET);
_e51(CLK := INST8.Q);
INST10(IN := _e51.Q, PT := time4, ET => ET);
_e52(CLK := INST13.Q);
INST15(IN := _e52.Q, PT := time4, ET => ET);
_e53(CLK := INST16.Q);
INST17(IN := _e53.Q, PT := T#2s, ET => ET);
_e54(CLK := INST23.Q);
INST25(IN := _e54.Q, PT := time4, ET => ET);
_e55(CLK := INST28.Q);
INST30(IN := _e55.Q, PT := time4, ET => ET);
_e56(CLK := INST31.Q);
INST32(IN := _e56.Q, PT := T#2s, ET => ET);
_e57(CLK := INST36.Q);
INST37(IN := _e57.Q, PT := T#4s, ET => ET);
%MX62 := INST5.Q OR INST10.Q OR INST15.Q OR INST17.Q OR INST25.Q OR INST30.Q OR INST32.Q OR INST37.Q;
(* Rung L261 *)
%IX0.0.46 := INST20.Q;
(* Rung L262 *)
_e58(CLK := INST1.Q);
INST2(IN := _e58.Q, PT := T#3s, ET => ET);
_e59(CLK := INST26.Q);
INST27(IN := _e59.Q, PT := T#3s, ET => ET);
%MX63 := INST2.Q OR INST27.Q;
(* Rung L269 *)
_e60(CLK := INST11.Q);
INST12(IN := _e60.Q, PT := T#3s, ET => ET);
_e61(CLK := INST33.Q);
INST34(IN := _e61.Q, PT := T#3s, ET => ET);
%MX49 := INST12.Q OR INST34.Q;

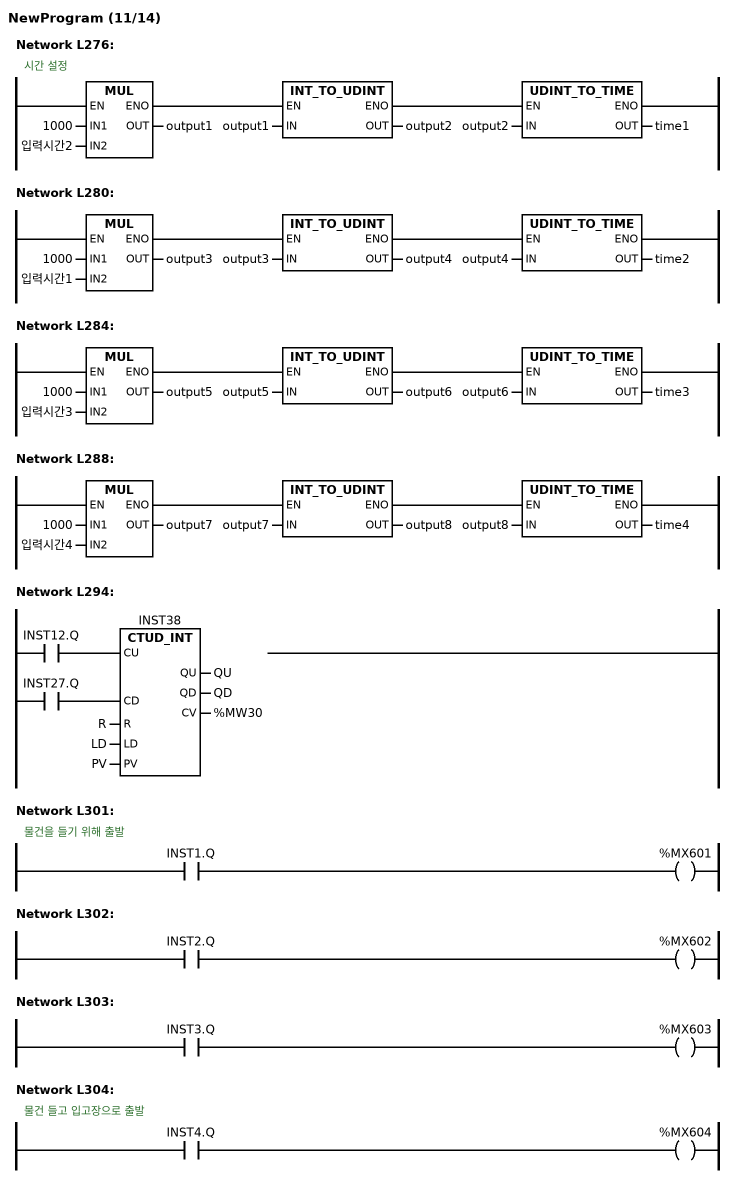
(* 시간 설정 *)
(* Rung L276 *)
output1 := 1000 * 입력시간2;
output2 := INT_TO_UDINT(output1);
time1 := UDINT_TO_TIME(output2);
(* Rung L280 *)
output3 := 1000 * 입력시간1;
output4 := INT_TO_UDINT(output3);
time2 := UDINT_TO_TIME(output4);
(* Rung L284 *)
output5 := 1000 * 입력시간3;
output6 := INT_TO_UDINT(output5);
time3 := UDINT_TO_TIME(output6);
(* Rung L288 *)
output7 := 1000 * 입력시간4;
output8 := INT_TO_UDINT(output7);
time4 := UDINT_TO_TIME(output8);
(* Rung L294 *)
INST38(CU := INST12.Q, CD := INST27.Q, R := R, LD := LD, PV := PV, QU => QU, QD => QD, CV => %MW30);
(* Rung L301 *)
%MX601 := INST1.Q;
(* 물건을 들기 위해 출발 *)
(* Rung L302 *)
%MX602 := INST2.Q;
(* Rung L303 *)
%MX603 := INST3.Q;
(* Rung L304 *)
%MX604 := INST4.Q;
(* 물건 들고 입고장으로 출발 *)

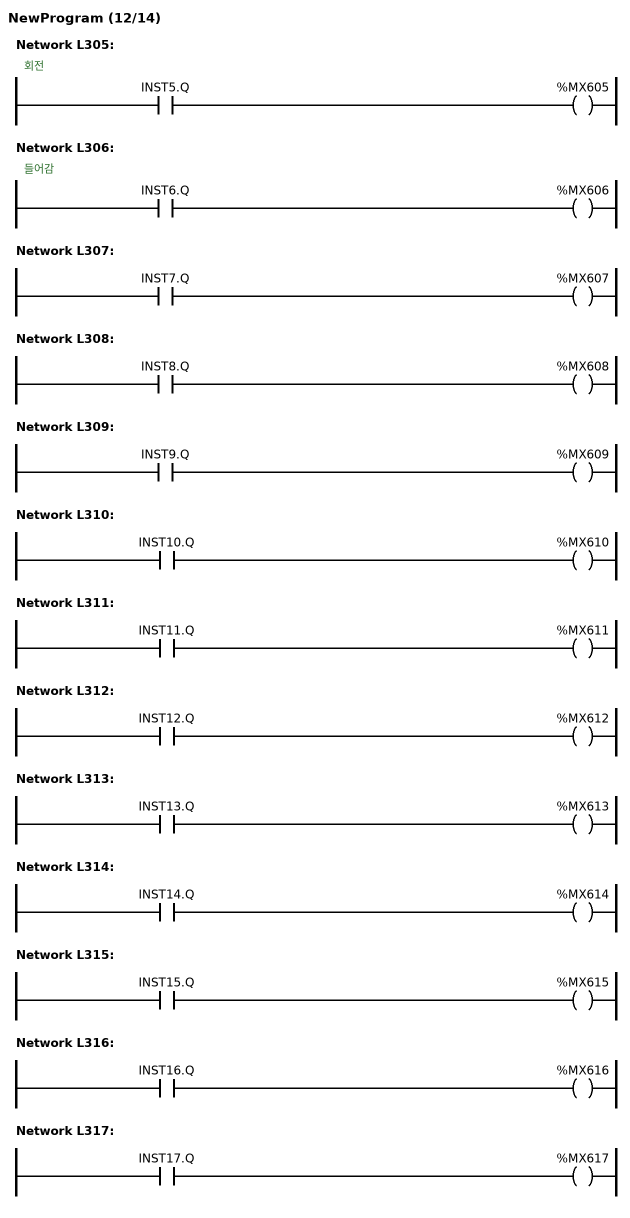
(* Rung L305 *)
%MX605 := INST5.Q;
(* 회전 *)
(* Rung L306 *)
%MX606 := INST6.Q;
(* 들어감 *)
(* Rung L307 *)
%MX607 := INST7.Q;
(* Rung L308 *)
%MX608 := INST8.Q;
(* Rung L309 *)
%MX609 := INST9.Q;
(* Rung L310 *)
%MX610 := INST10.Q;
(* Rung L311 *)
%MX611 := INST11.Q;
(* Rung L312 *)
%MX612 := INST12.Q;
(* Rung L313 *)
%MX613 := INST13.Q;
(* Rung L314 *)
%MX614 := INST14.Q;
(* Rung L315 *)
%MX615 := INST15.Q;
(* Rung L316 *)
%MX616 := INST16.Q;
(* Rung L317 *)
%MX617 := INST17.Q;

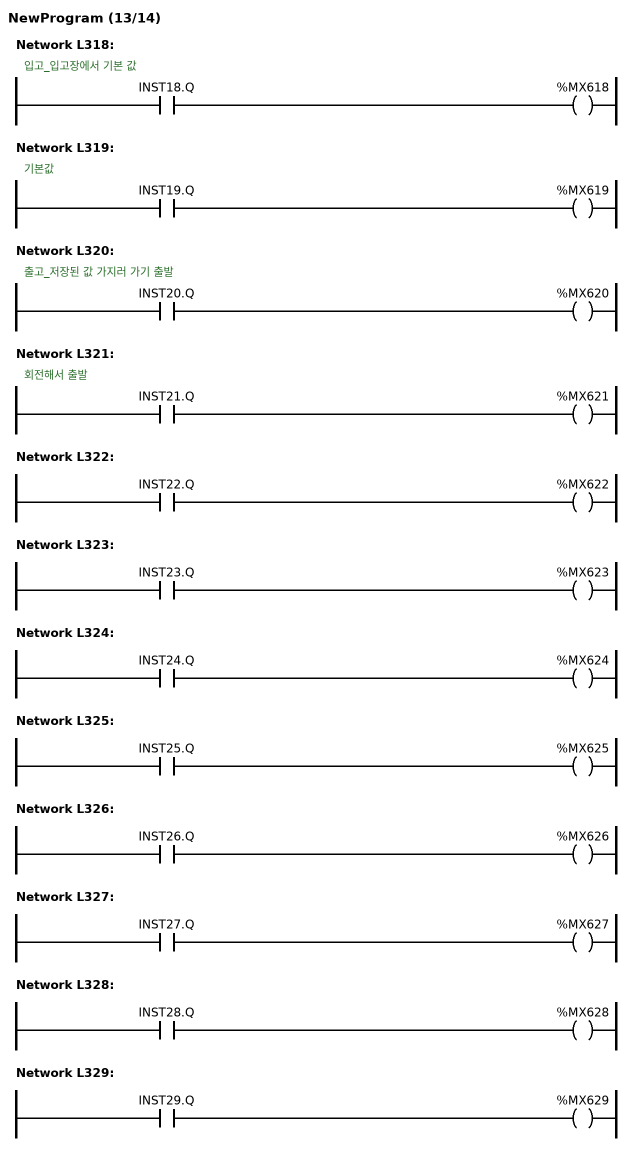
(* Rung L318 *)
%MX618 := INST18.Q;
(* 입고_입고장에서 기본 값 *)
(* Rung L319 *)
%MX619 := INST19.Q;
(* 기본값 *)
(* Rung L320 *)
%MX620 := INST20.Q;
(* 출고_저장된 값 가지러 가기 출발 *)
(* Rung L321 *)
%MX621 := INST21.Q;
(* 회전해서 출발 *)
(* Rung L322 *)
%MX622 := INST22.Q;
(* Rung L323 *)
%MX623 := INST23.Q;
(* Rung L324 *)
%MX624 := INST24.Q;
(* Rung L325 *)
%MX625 := INST25.Q;
(* Rung L326 *)
%MX626 := INST26.Q;
(* Rung L327 *)
%MX627 := INST27.Q;
(* Rung L328 *)
%MX628 := INST28.Q;
(* Rung L329 *)
%MX629 := INST29.Q;

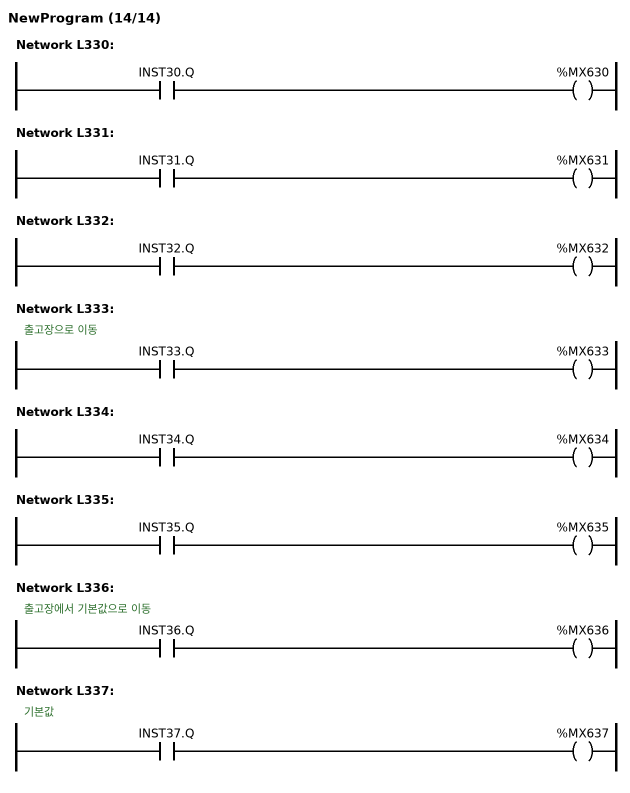
(* Rung L330 *)
%MX630 := INST30.Q;
(* Rung L331 *)
%MX631 := INST31.Q;
(* Rung L332 *)
%MX632 := INST32.Q;
(* Rung L333 *)
%MX633 := INST33.Q;
(* 출고장으로 이동 *)
(* Rung L334 *)
%MX634 := INST34.Q;
(* Rung L335 *)
%MX635 := INST35.Q;
(* Rung L336 *)
%MX636 := INST36.Q;
(* 출고장에서 기본값으로 이동 *)
(* Rung L337 *)
%MX637 := INST37.Q;
(* 기본값 *)
END_PROGRAM